// TwinCAT 3 PLC project Untitled1
// ProgramVersion: 3.1.4023.0
// libraries:
//   Tc2_Standard, * (Beckhoff Automation GmbH)
//   Tc2_System, * (Beckhoff Automation GmbH)
//   Tc3_Module, * (Beckhoff Automation GmbH)
// project tree:
//   DUTs/ DropdownBox.TcDUT
//   / PlcTask.TcTTO
//   POUs/ MAIN.TcPOU
// real-time tasks:
//   TASK PlcTask: cycle T#10ms, priority 20, ADS port 350

CONFIGURATION Untitled1
    RESOURCE PLC ON TwinCAT3
        TASK PlcTask(INTERVAL := T#10ms, PRIORITY := 20);
        PROGRAM MAIN WITH PlcTask : MAIN;
    END_RESOURCE
END_CONFIGURATION

// ---- DUTs/DropdownBox.TcDUT
{attribute 'qualified_only'}
{attribute 'strict'}
TYPE DropdownBox :
(
	first_page,
	Second_page
);
END_TYPE

// ---- POUs/MAIN.TcPOU
PROGRAM MAIN
VAR
	test : STRING := 'hello'; //this is a test variable to place in the textbox on the HMI
	//SAFE
	HoldButton : BOOL := FALSE;
	HoldSwitchLight : BOOL;
	SwitchButton : BOOL := FALSE;
	SwitchButtonLight : BOOL;
	
	StopButton : BOOL;
	StartButton : BOOL;

	Options : DropdownBox;
	
	bProcess_Status:BOOL;//the timer light
	tProcess_Duration:TIME;
	fbProcess_Timer:TON;
	bTimer_Done:BOOL;
END_VAR

fbProcess_Timer(IN:= bProcess_Status,PT:=tProcess_Duration ,Q=> bTimer_Done,ET=> );

HoldSwitchLight:=HoldButton;
SwitchButtonLight:=SwitchButton;

IF StartButton THEN
	bProcess_Status:=TRUE;
END_IF

IF StopButton OR bTimer_Done THEN
	bProcess_Status:=FALSE;
	//HoldButton:=FALSE;
	SwitchButton:=FALSE;
END_IF

END_PROGRAM
